(*
  Base camera system
  Implements I_Camera: set I_CameraSink.   
*)
FUNCTION_BLOCK ABSTRACT FB_CameraBase EXTENDS FB_Commons IMPLEMENTS I_Camera, I_CameraTriggerDevice

VAR
  _bInitialized             : BOOL;
  _iCameraSink              : I_CameraSink;
  _iCameraTrigger           : I_CameraTrigger;
  _bSimulate                : BOOL;
  _nPrintUnitResolution     : UDINT;           (*printhead pixel resolution [dpi]*)
  _nPrintUnitSubPx          : UDINT;           (*print unit SubPixel resolution [SubPx]*)
  _bUseCameraTrigger        : BOOL;            (*use a trigger output timestamp I/O*)
  _bUseCameraTriggerFeedback : BOOL;           (*use a camera triggered feedback timestamp I/O*)
  _eCameraMode              : E_CameraMode;    (*desired camera mode*)
  _ePossibleMode            : E_CameraMode;    (*currently possible mode*)
  _fSubstrateLength         : LREAL := 1;      (*Substrate length [m]*)
  _fSubstrateWidth          : LREAL := 1;      (*Substrate width [m]*)
  _fImageLength             : LREAL := 1;      (*Image length [m]*)
  _fImageWidth              : LREAL := 1;      (*Image width [m]*)
  _fFrameLength             : LREAL := 1;      (*Camera Frame width in [px]*)
  _bActivated               : BOOL;
  _sVisuName                : STRING := 'unvailable';     (*detail visualisation instance name*)
  _nRxCamPoints             : UDINT;                      (*number of received cam points*)
  stCamPoint                : ST_DeformationPointAccurate;(*actual camera point*)
  
  _bCamTriggerOk            : BOOL;
  _bCamStarted              : BOOL;
  _bCamDone                 : BOOL;   
  _nCamStartPos             : DINT;    //Cam start position ideal [SubPx]
  _nCamStartPosDeviation    : DINT;    //Cam stated position real [SubPx]
  
  // messaging
  _pMsgConfig               : POINTER TO CalmarCommons.ST_MSG_CONFIG;
END_VAR

VAR PERSISTENT
  _fTriggerDistance         : LREAL;           (*Distance between Sensor and Trigger [m]*)
  _fTriggerPulseLength      : LREAL := 10;     (*Length of trigger signal in ms, min. 3 bus cycles*)
  _fDetectToCameraOffset    : LREAL := 0.1;    (*Distance between innput trigger and camera, mech.*)
  _fCameraToPrintOffset     : LREAL := 0.0;    (*Distance between Camera and PU, mech, This offset can be used to shift the reference of a camera/sheet-detect, e.g. because this reference is different from to one where the alignment Camera/sheetdetect-PrintUnit has been made*)
END_VAR

METHOD ActivateCam : BOOL
VAR_INPUT
  iCameraSink : I_CameraSink;
END_VAR
IF iCameraSink = 0 THEN
  LogError('Invalid parameter (0 pointer)');
  ActivateCam := FALSE;
  RETURN; 
ELSIF _iCameraSink <> 0 AND iCameraSink <>_iCameraSink THEN
  LogError('SetSink failed: other sink already exists');
  ActivateCam := FALSE;
  RETURN; 
END_IF 

_iCameraSink := iCameraSink;
_iCameraTrigger.Enable(iCam := THIS^,bUseCameraTrigger:= _bUseCameraTrigger, bUseCameraTriggerFeedback:=_bUseCameraTriggerFeedback);

_bActivated := TRUE;
ActivateCam:=TRUE;
END_METHOD

(*
  Activate/Deactivate camera trigger device
*)
PROPERTY bEnableTrigger : BOOL
SET
IF bEnableTrigger THEN
  _iCameraTrigger.Enable(iCam := THIS^, bUseCameraTrigger:= _bUseCameraTrigger, bUseCameraTriggerFeedback:=_bUseCameraTriggerFeedback);
ELSE
  _iCameraTrigger.Disable();
END_IF
END_SET
END_PROPERTY

(*
  Activate/Deactivate camera manual teach mode
*)
PROPERTY bManualTeach : BOOL
SET
_iCameraTrigger.bManualTeach := bManualTeach;
END_SET
END_PROPERTY

{attribute 'monitoring':='call'}
PROPERTY bSimulate : BOOL
GET
bSimulate := _bSimulate;
END_GET
SET
_bSimulate := bSimulate;
END_SET
END_PROPERTY

METHOD CamTrigger
VAR_INPUT
  bOk             : BOOL;     // trigger is ok
	nPos            : DINT;     // camera triggered position
  nPosDeviation   : DINT;     // camera started deviation
END_VAR
_nRxCamPoints := 0;
_bCamStarted    := TRUE;
_bCamDone       := FALSE;
_bCamTriggerOk  := bOk;
_nCamStartPos   := nPos;
_nCamStartPosDeviation := nPosDeviation;

IF _iCameraSink <> 0 THEN   // link to sink (wokerCam -> CT)
  ;
END_IF
END_METHOD

METHOD CamTriggerDone
_bCamStarted    := FALSE;  // this call marks the end of the camera trigger period
_bCamDone       := TRUE;
END_METHOD

METHOD DeactivateCam : BOOL
VAR_INPUT
  iSink : I_CameraSink;
END_VAR
IF _iCameraSink <> 0 AND iSink <> _iCameraSink THEN
  LogError('remove sink failed: inconsistent');
  DeactivateCam := FALSE;
  RETURN;  
END_IF

_iCameraSink := 0;
_iCameraTrigger.Disable();
_bActivated := FALSE;
DeactivateCam:=TRUE;
END_METHOD

{attribute 'monitoring':='call'}
PROPERTY ABSTRACT eCameraMode : E_CameraMode
GET
END_GET
END_PROPERTY

{attribute 'monitoring':='call'}
PROPERTY ABSTRACT eDeviceType : E_CameraDevice
GET
END_GET
END_PROPERTY

{attribute 'monitoring':='call'}
PROPERTY fCameraToPrintOffset : LREAL
GET
//This offset can be used to shift the reference of a camera, e.g. because this reference is different from to one where the alignment Camera-PrintUnit has been made
fCameraToPrintOffset := _fCameraToPrintOffset;
END_GET
SET
_fCameraToPrintOffset := fCameraToPrintOffset;
END_SET
END_PROPERTY

{attribute 'monitoring':='call'}
PROPERTY fDetectToCameraOffset : LREAL
GET
//This offset can be used to shift the reference of a camera, e.g. because this reference is different from to one where the alignment Camera-PrintUnit has been made
fDetectToCameraOffset := _fDetectToCameraOffset;
END_GET
SET
_fDetectToCameraOffset := fDetectToCameraOffset;
END_SET
END_PROPERTY

{attribute 'monitoring':='call'}
(* camera frame size in [px]*)
PROPERTY fFrameLength : LREAL
GET
fFrameLength := _fFrameLength;
END_GET
SET
_fFrameLength := fFrameLength;
END_SET
END_PROPERTY

{attribute 'monitoring':='call'}
(*Image Length/Depth in [m]*)
PROPERTY fImageLength : LREAL
GET
fImageLength := _fImageLength;
END_GET
SET
_fImageLength := fImageLength;
END_SET
END_PROPERTY

{attribute 'monitoring':='call'}
(*Image Width in [m]*)
PROPERTY fImageWidth : LREAL
GET
fImageWidth := _fImageWidth;
END_GET
SET
_fImageWidth := fImageWidth;
END_SET
END_PROPERTY

{attribute 'monitoring':='call'}
(*Substrate Length/Depth in [m]*)
PROPERTY fSubstrateLength : LREAL
GET
fSubstrateLength := _fSubstrateLength;
END_GET
SET
//ROI in Print direction
IF _iCameraTrigger <> 0 THEN
  _iCameraTrigger.SetSubstrateLength(fSubstrateLength := fSubstrateLength);   // save to camera trigger
  _fSubstrateLength := fSubstrateLength;                                      // save to camera
END_IF
END_SET
END_PROPERTY

{attribute 'monitoring':='call'}
(*Substrate Width in [m]*)
PROPERTY fSubstrateWidth : LREAL
GET
fSubstrateWidth := _fSubstrateWidth;
END_GET
SET
_fSubstrateWidth := fSubstrateWidth;
END_SET
END_PROPERTY

{attribute 'monitoring':='call'}
PROPERTY fTriggerDistance : LREAL
GET
fTriggerDistance := _fTriggerDistance;
END_GET
SET
_fTriggerDistance := fTriggerDistance;
END_SET
END_PROPERTY

PROPERTY fTriggerPulseLength : LREAL
GET
fTriggerPulseLength := _fTriggerPulseLength;
END_GET
END_PROPERTY

METHOD ABSTRACT GetCamState : BOOL
VAR_OUTPUT
  bCamModeNotSupported  : BOOL;   // desired camera mode not supported
  bCam
END_VAR
END_METHOD

METHOD ABSTRACT GetCamStatus : BOOL
VAR_OUTPUT
  bConnectionOK  : BOOL;    // Camera connected
  bTeachOk       : BOOL;    // Teach successful
  nTeachedPoints : UDINT;   // Teached points for this job
  nScannedPoints : UDINT;   // Scanned points on current sheet  
  bCamStarted    : BOOL;    // Camera trigger is active, cam started
  bCamDone       : BOOL;    // Camera finished on last CT
  bErrors        : ARRAY[1..GVL_Camera.nC_NbCamErrors] OF BOOL;  // generic error flag list
END_VAR
END_METHOD

METHOD Init
VAR_INPUT
  nPrintUnitResolution         : UDINT;    (*printhead pixel resolution [dpi]*)
  nPrintUnitSubPx              : UDINT;    (*print unit subPixel resolution [SubPx]*)
  iCameraTrigger               : I_CameraTrigger;
  bUseCameraTrigger            : BOOL;     (*use a trigger output timestamp I/O*)
  bUseCameraTriggerFeedback    : BOOL;     (*use a camera triggered feedback timestamp I/O*)
END_VAR
IF nPrintUnitResolution <> 0 AND iCameraTrigger <> 0 THEN
  _nPrintUnitResolution := nPrintUnitResolution;
  _nPrintUnitSubPx      := nPrintUnitSubPx;
  _iCameraTrigger       := iCameraTrigger;
  
  _bUseCameraTrigger := bUseCameraTrigger;
  _bUseCameraTriggerFeedback := bUseCameraTriggerFeedback;
  
  _bInitialized := TRUE;
ELSE
  _bInitialized := FALSE;
END_IF
END_METHOD

METHOD mJobStart : BOOL
END_METHOD

(*
  Set mode to camera.
  :return: TRUE if success
*)
METHOD ABSTRACT setCameraMode : BOOL
VAR_INPUT
  eCameraMode : E_CameraMode;
END_VAR
END_METHOD

METHOD setMsgInterface : BOOL
VAR_INPUT
	pMsgConfig	: POINTER TO CalmarCommons.ST_MSG_CONFIG;
END_VAR
_pMsgConfig := pMsgConfig;
END_METHOD

{attribute 'monitoring':='call'}
PROPERTY sName : STRING
GET
sName := 'undefined';
END_GET
END_PROPERTY

{attribute 'monitoring':='call'}
PROPERTY sVisuName : STRING
GET
sVisuName := _sVisuName;
END_GET
SET
_sVisuName := sVisuName;
END_SET
END_PROPERTY

END_FUNCTION_BLOCK

(* stored: Version 1.1.0.1, ProductVersion 3.1.4024.3
   POU FB_CameraBase: Id {484ed993-7aea-449c-8988-777e097fbb7c}, SpecialFunc None
   Method ActivateCam: Id {e847224c-0022-43ce-b368-4855714fcc0c}
   Property bEnableTrigger: Id {26714317-df55-4926-95ca-e8d277e6a9f4}
   Set Set: Id {71545a42-507c-4010-a44b-2af7d6ec7ab1}
   Property bManualTeach: Id {7c1a0e8e-c614-4379-bba3-244c737d9b61}
   Set Set: Id {4c52ff0d-ffde-43a5-806a-9464789b6fa0}
   Property bSimulate: Id {d4820fc1-ed9d-464e-80c6-eee254d40168}
   Get Get: Id {38619303-c217-4e7d-b79e-7fac24a44719}
   Set Set: Id {fbd6b5ab-08b4-4f62-a0ad-b03e1ee0d1be}
   Method CamTrigger: Id {42261f93-e978-469f-9dd2-7f31b656b223}
   Method CamTriggerDone: Id {64c1da17-4b35-43a3-b060-9ad844c6ae65}
   Method DeactivateCam: Id {925d77c2-f95c-4f3d-a4ef-64648960cc56}
   Property eCameraMode: Id {b13f5b24-e0b7-48dd-97dd-ad6fa7e18f64}
   Get Get: Id {2c312843-8d5b-482a-9c83-bd1bdd0999e0}
   Property eDeviceType: Id {94438f1e-950c-467e-8969-b0c0d5a5f856}
   Get Get: Id {06377dc2-6bfa-4388-8a9e-9bcbd62af831}
   Property fCameraToPrintOffset: Id {093fd995-ed0b-4047-aa59-b89332069d30}
   Get Get: Id {8ee24d4f-0fab-4aec-bb70-683f0e6fdb78}
   Set Set: Id {763d1dcf-b230-441d-be7d-93610dfaea41}
   Property fDetectToCameraOffset: Id {c3ef6c91-7f21-478d-9985-2a721dd9979b}
   Get Get: Id {fbb051dc-3e60-4957-a891-17005f99ce6f}
   Set Set: Id {8111f578-f7b5-4695-87cd-ac5b7998e7cd}
   Property fFrameLength: Id {2fe04168-73eb-400e-9296-7718ae9f89f9}
   Get Get: Id {e75e4fb9-0624-4cb2-9591-13fb0dea9607}
   Set Set: Id {fcbedb1b-8417-42d9-8178-0d96c0ed5e77}
   Property fImageLength: Id {e37bb5ee-3065-4a07-876d-1955a6190a4c}
   Get Get: Id {79bce027-86cf-4668-a756-af0c31abec21}
   Set Set: Id {338fc4be-632a-4746-ac96-467b1e71a90e}
   Property fImageWidth: Id {09d6d256-6435-4243-8305-b72f057cdfe5}
   Get Get: Id {7a6663f4-cb8d-4a12-b0db-930f57ab1d63}
   Set Set: Id {ebfa97bf-e36e-4c70-a87b-13c1cdc2794e}
   Property fSubstrateLength: Id {39d153bb-814c-429f-938c-0b96b9603b8b}
   Get Get: Id {ecc44cd6-f328-4fb0-bcff-3a6a6e7bb9ed}
   Set Set: Id {e2925e44-fa5a-4283-8bb7-8311068c3698}
   Property fSubstrateWidth: Id {490a4387-df1e-483d-a915-be97914a0a12}
   Get Get: Id {6278d786-89e3-49db-886a-4543ba2f5070}
   Set Set: Id {ec4eda75-b3a1-4038-80d8-8830e633b225}
   Property fTriggerDistance: Id {f65a3627-7304-49e3-921f-3161a7b67530}
   Get Get: Id {0ff07811-262e-43d1-b963-3df0600f9e55}
   Set Set: Id {72254900-a7b6-48a8-a8e1-245044b91966}
   Property fTriggerPulseLength: Id {5efe63ba-d1b7-4c49-b79b-6cfc9d271b93}
   Get Get: Id {b94ca0d1-d3c4-4849-94e1-ff9e65038505}
   Method GetCamState: Id {17117628-5115-49f0-8f45-ad0bb105b7ac}
   Method GetCamStatus: Id {2f1b9c70-d6ea-4216-8ad6-ef84259fa168}
   Method Init: Id {7a74c0b9-9e9e-4d88-9483-cf9903fb3814}
   Method mJobStart: Id {21a24940-50c3-4289-8331-b554488b8e7f}
   Method setCameraMode: Id {f64e889a-3cd6-467f-aad2-c7d8acb483a7}
   Method setMsgInterface: Id {7dd5c4d3-99b2-4cc8-98b5-88572882d484}
   Property sName: Id {b16fccb6-779e-42b9-bde6-87fe58d4f1e1}
   Get Get: Id {a6f60ccd-169f-456f-aae0-4ff0b379c6be}
   Property sVisuName: Id {b120037b-3d94-4baa-bd12-ddb399b9e512}
   Get Get: Id {4e8511df-8759-4687-aad0-92498953e579}
   Set Set: Id {3bdd9c08-3ac1-46df-9f4f-63b614ba4637} *)
